// TIA Portal V21 export
FUNCTION "Motore_PompaOlio" : Void   // FC129, LAD
{ S7_Optimized_Access := 'TRUE' }
// stored: SetENOAutomatically false
   VAR_TEMP
      AutoPos : Bool;
      AutoNeg : Bool;
   END_VAR
BEGIN

REGION Network 1: Comando positivo in automatico
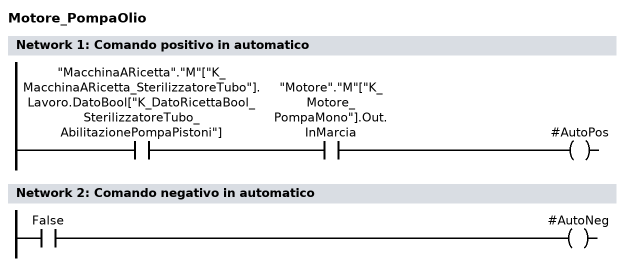
   RUNG wire#powerrail
      Contact( "MacchinaARicetta"."M"["K_MacchinaARicetta_SterilizzatoreTubo"].Lavoro.DatoBool["K_DatoRicettaBool_SterilizzatoreTubo_AbilitazionePompaPistoni"] )
      Contact( "Motore"."M"["K_Motore_PompaMono"].Out.InMarcia )
      Coil( #AutoPos )
   END_RUNG
   // the same network as SCL:
   #AutoPos := "MacchinaARicetta"."M"["K_MacchinaARicetta_SterilizzatoreTubo"].Lavoro.DatoBool["K_DatoRicettaBool_SterilizzatoreTubo_AbilitazionePompaPistoni"] AND "Motore"."M"["K_Motore_PompaMono"].Out.InMarcia;
END_REGION

REGION Network 2: Comando negativo in automatico
   RUNG wire#powerrail
      Contact( False )
      Coil( #AutoNeg )
   END_RUNG
   // the same network as SCL:
   #AutoNeg := False;
END_REGION

REGION Network 3 (SCL)
   REGION AgitatoreVascaProdotto
       REGION Ingressi
           "Motore".M[K_Motore_PompaOlio].In.FbDigitali.TermicoIntervenuto := NOT "PompaOlio_TermicoOk";
           "Motore".M[K_Motore_PompaOlio].In.FbDigitali.FeedbackMarcia := "PompaOlio_Marcia";
           "Motore".M[K_Motore_PompaOlio].In.CmdPosRich := #AutoPos;
           "Motore".M[K_Motore_PompaOlio].In.CmdNegRich := #AutoNeg;
       END_REGION ;
       REGION Gestione
           "GestMotore"(K_Motore := "K_Motore_PompaOlio",
                        K_TipoMotore := "K_TipoMotore_Teleruttore2Dir",
                        K_Zona := "K_Zona_Sterilizzatore");
       END_REGION ;
       REGION Uscite
           "PompaOlio_ComandoMarcia" := "Motore".M[K_Motore_PompaOlio].Out.CmdPosMotore;
       END_REGION ;
   END_REGION ;
END_REGION
END_FUNCTION
